(* IEC 61131-3 sources: ATCMcontrol_Engineering/src/Target/ATHW119/Libs/ATCM_IEC1131_3/table_28, 6 files *)

(* ---- eq.st ---- *)
(*[[
    UserURL= "ATCMfile:EQ.htm"
]]*)

FUNCTION EQ : BOOL
VAR_INPUT
    IN1 : ANY_ELEMENTARY;
END_VAR
VAR_IN_EXT
    IN2 : ANY_ELEMENTARY;
END_VAR

inline =

END_FUNCTION

(* ---- ge.st ---- *)
(*[[
    UserURL= "ATCMfile:GE.htm"
]]*)

FUNCTION GE : BOOL
VAR_INPUT
    IN1 : ANY_ELEMENTARY;
END_VAR
VAR_IN_EXT
    IN2 : ANY_ELEMENTARY;
END_VAR

inline >=

END_FUNCTION

(* ---- gt.st ---- *)
(*[[
    UserURL= "ATCMfile:GT.htm"
]]*)

FUNCTION GT : BOOL
VAR_INPUT
    IN1 : ANY_ELEMENTARY;
END_VAR
VAR_IN_EXT
    IN2 : ANY_ELEMENTARY;
END_VAR

inline >

END_FUNCTION

(* ---- le.st ---- *)
(*[[
    UserURL= "ATCMfile:LE.htm"
]]*)

FUNCTION LE : BOOL
VAR_INPUT
    IN1 : ANY_ELEMENTARY;
END_VAR
VAR_IN_EXT
    IN2 : ANY_ELEMENTARY;
END_VAR

inline <=

END_FUNCTION

(* ---- lt.st ---- *)
(*[[
    UserURL= "ATCMfile:LT.htm"
]]*)

FUNCTION LT : BOOL
VAR_INPUT
    IN1 : ANY_ELEMENTARY;
END_VAR
VAR_IN_EXT
    IN2 : ANY_ELEMENTARY;
END_VAR

inline <

END_FUNCTION

(* ---- ne.st ---- *)
(*[[
    UserURL= "ATCMfile:NE.htm"
]]*)

FUNCTION NE : BOOL
VAR_INPUT
    IN1 : ANY_ELEMENTARY;
    IN2 : ANY_ELEMENTARY;
END_VAR

inline <>

END_FUNCTION
